FUNCTION Simula_Compila_Mis 
VAR_INPUT
	auxMis   : REFERENCE TO MIS_PC;
END_VAR
VAR
	ni	: UINT :=0;
END_VAR

//----------------------------------------------------
// Simula Creazione Missione
// Elaborata impulsivamente compila la missione        
//----------------------------------------------------
auxMis.Pstart_PC		:=143;
auxMis.PEnd_PC			:=175;
auxMis.Typ_car_PC		:=0;		// stabilità max
//------------------ 1
ni := ni + 1;
auxMis.Step_PC[ni].ps 	:= 144;
auxMis.Step_PC[ni].dist := 100;
auxMis.Step_PC[ni].Comandi.In_Mov_Y 	:= TRUE;
auxMis.Step_PC[ni].Comandi.In_Mov_Av 	:= TRUE;
auxMis.Step_PC[ni].Comandi.Lenta 		:= TRUE;	// cambio corsia
//------------------ 2
ni := ni + 1;
auxMis.Step_PC[ni].ps 	:= 154;
auxMis.Step_PC[ni].dist := 100;
auxMis.Step_PC[ni].Comandi.In_Mov_X 	:= TRUE;
auxMis.Step_PC[ni].Comandi.In_Mov_Av 	:= TRUE;
//------------------ 3
ni := ni + 1;
auxMis.Step_PC[ni].ps 	:= 164;
auxMis.Step_PC[ni].dist := 100;
auxMis.Step_PC[ni].Comandi.In_Mov_X 	:= TRUE;
auxMis.Step_PC[ni].Comandi.In_Mov_Av 	:= TRUE;
//------------------ 4
ni := ni + 1;
auxMis.Step_PC[ni].ps 	:= 174;
auxMis.Step_PC[ni].dist := 100;
auxMis.Step_PC[ni].Comandi.In_Mov_X 	:= TRUE;
auxMis.Step_PC[ni].Comandi.In_Mov_Av 	:= TRUE;
//------------------ 5
ni := ni + 1;
auxMis.Step_PC[ni].ps 	:= 175;
auxMis.Step_PC[ni].dist := 100;
auxMis.Step_PC[ni].Comandi.In_Mov_Y 	:= TRUE;
auxMis.Step_PC[ni].Comandi.In_Mov_Av 	:= TRUE;
auxMis.Step_PC[ni].Comandi.Lenta 		:= TRUE;	// cambio corsia
//------------------ 6
ni := ni + 1;
auxMis.Step_PC[ni].ps 	:= 175;
auxMis.Step_PC[ni].dist := 0;						// carico su stesso nodo 175
auxMis.Step_PC[ni].Comandi.CarSoll_0 	:= TRUE;	// carico
//------------------ 7
ni := ni + 1;
auxMis.Step_PC[ni].ps 	:= 175;
auxMis.Step_PC[ni].dist := 0;				// fine miss su stesso nodo 175
auxMis.Step_PC[ni].Comandi.End 	:= TRUE;	// fine miss
//------------------ 
auxMis.Tot_Step_PC	:=ni;					// nr. Tot Step

END_FUNCTION

(* stored: Version 1.1.0.1, ProductVersion 3.1.4024.11
   POU Simula_Compila_Mis: Id {c6d656b8-5506-4a96-9351-36f84dcd939d}, SpecialFunc None *)
